FUNCTION_BLOCK "Semantic_AnyInOutput"
{ S7_Optimized_Access := 'TRUE' }
VERSION : 0.1

VAR_OUTPUT
    badAny : Any;
    // EXPECT: error[type.illegal-section] SEM-SECTION-002
END_VAR

BEGIN
END_FUNCTION_BLOCK
